FUNCTION_BLOCK SS2 (* Composite FB wrapping other FBs *)
  (* Standard: 61499-2 *)
  (* Version 1.0, 2024-08-30, DEVIASH *)
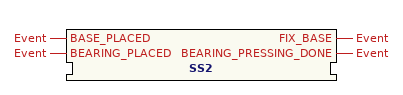
  EVENT_INPUT
    BASE_PLACED; (* Initialization Request *)
    BEARING_PLACED;
  END_EVENT
  EVENT_OUTPUT
    FIX_BASE; (* Initialization Confirm *)
    BEARING_PRESSING_DONE;
  END_EVENT
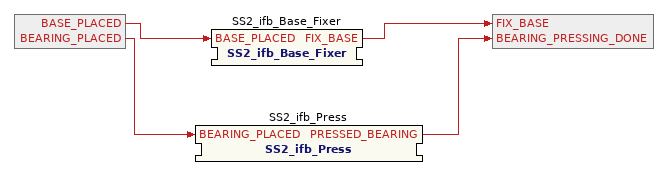
  FBS
    SS2_ifb_Base_Fixer : SS2_ifb_Base_Fixer;
    SS2_ifb_Press : SS2_ifb_Press;
  END_FBS
  EVENT_CONNECTIONS
    BASE_PLACED TO SS2_ifb_Base_Fixer.BASE_PLACED;
    SS2_ifb_Base_Fixer.FIX_BASE TO FIX_BASE;
    BEARING_PLACED TO SS2_ifb_Press.BEARING_PLACED;
    SS2_ifb_Press.PRESSED_BEARING TO BEARING_PRESSING_DONE;
  END_CONNECTIONS
END_FUNCTION_BLOCK
